// TIA Portal V18 export
FUNCTION_BLOCK "_hmi_singleSpotManager"   // FB59, FBD
{ S7_Optimized_Access := 'TRUE' }
VERSION : 0.1
// stored: AutoNumber true, IsIECCheckEnabled false, IsRetainMemResEnabled false, MemoryReserve 100, SetENOAutomatically false, UDAEnableTagReadback false
   VAR_INPUT
      hmi_PosSet : "typePositions";
      cur_pos_set : "typePositions";
   END_VAR
   VAR_IN_OUT
      hmiFromHmi : Bool;
      hmiSFromEncoder : Bool;
      posToModify : "typePositions";
   END_VAR
   VAR
      N_max : Int := 99;
   END_VAR
BEGIN

REGION Network 1
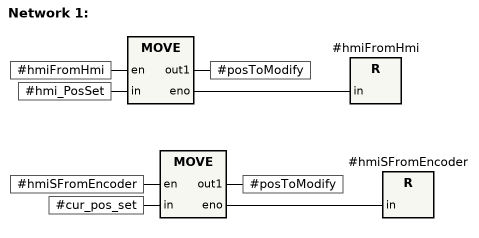
   IF #hmiFromHmi THEN
       #posToModify := #hmi_PosSet;
       #hmiFromHmi := FALSE;
   END_IF;
   IF #hmiSFromEncoder THEN
       #posToModify := #cur_pos_set;
       #hmiSFromEncoder := FALSE;
   END_IF;
END_REGION
END_FUNCTION_BLOCK
